// TIA Portal V17 export
// export: Created 2024-10-17T14:16:12.2521247Z, ExportSetting WithDefaults, DisplayName Totally Integrated Automation Portal, DisplayVersion V17 Update 4, DisplayName TIA Portal Openness, DisplayVersion V17 Update 4, DisplayName TIA Portal Version Control Interface, DisplayVersion V17, DisplayName SINAMICS Startdrive Advanced, DisplayVersion V17 Update2, DisplayName SINAMICS Startdrive G130, G150, S120, S150, SINAMICS MV, S210, DisplayVersion V17 Update2, DisplayName SINAMICS Startdrive G110M, G120, G120C, G120D, G120P, G115D, DisplayVersion V17 Update2, DisplayName STEP 7 Professional, DisplayVersion V17 Update 4, DisplayName STEP 7 Safety, DisplayVersion V17, DisplayName WinCC Advanced / Unified PC, DisplayVersion V17 Update 4
ORGANIZATION_BLOCK "Main"   // OB1, LAD, ProgramCycle
TITLE = "Main Program Sweep (Cycle)"
{ S7_Optimized_Access := 'TRUE' }
VERSION : 0.1
// stored: AutoNumber true, IsIECCheckEnabled false, SetENOAutomatically false
   VAR_INPUT
      Initial_Call : Bool;   // Initial call of this OB
      Remanence : Bool;   // =True, if remanent data are available
   END_VAR
BEGIN

REGION Network 1: Example of calling LPMLV2022_UnitModeStateManager incl. ToDo structure
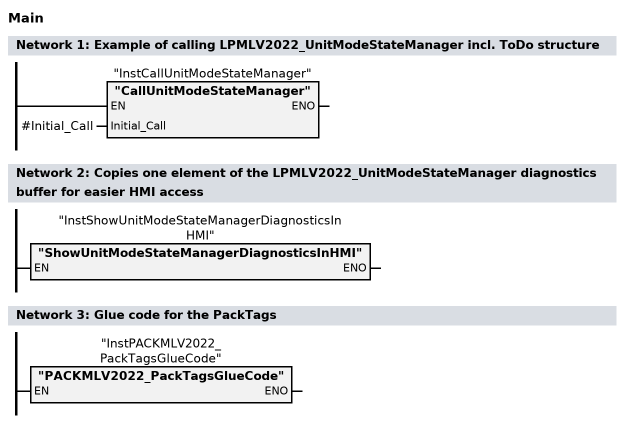
   RUNG wire#powerrail
      "InstCallUnitModeStateManager"(Initial_Call := #Initial_Call)
   END_RUNG
   // the same network as SCL:
   "InstCallUnitModeStateManager"(Initial_Call := #Initial_Call);   // "CallUnitModeStateManager"
END_REGION

REGION Network 2: Copies one element of the LPMLV2022_UnitModeStateManager diagnostics buffer for easier HMI access
   RUNG wire#powerrail
      "InstShowUnitModeStateManagerDiagnosticsInHMI"()
   END_RUNG
   // the same network as SCL:
   "InstShowUnitModeStateManagerDiagnosticsInHMI"();   // "ShowUnitModeStateManagerDiagnosticsInHMI"
END_REGION

REGION Network 3: Glue code for the PackTags
   RUNG wire#powerrail
      "InstPACKMLV2022_PackTagsGlueCode"()
   END_RUNG
   // the same network as SCL:
   "InstPACKMLV2022_PackTagsGlueCode"();   // "PACKMLV2022_PackTagsGlueCode"
END_REGION
END_ORGANIZATION_BLOCK
